TYPE EM_Transport_Mechanische_Stop_WRN :
STRUCT
END_STRUCT
END_TYPE

(* stored: Version 1.1.0.1, ProductVersion 3.1.4024.12
   DUT EM_Transport_Mechanische_Stop_WRN: Id {9f831520-7174-4c9c-a876-d34c3ed3af63} *)
